{attribute 'qualified_only'}
{attribute 'strict'}
TYPE AutostoreControlCommand :
(
	DO_NOTHING := 0,
	START	:= 1,
	STOP	:= 2
);
END_TYPE

(* stored: Version 1.1.0.1, ProductVersion 3.1.4024.12
   DUT AutostoreControlCommand: Id {7d13ff55-fc6b-4881-aa3a-15c0dcc71b09} *)
